(* IEC 61131-3 sources: robocpp/crates/iec_language_service/tests/fixtures, 1 file *)

(* ---- counter.st ---- *)
PROGRAM Counter
VAR
    Count : INT := 0;
END_VAR
Count := Count + 1;
END_PROGRAM
